INTERFACE INTERNAL I_StateInternal

PROPERTY INTERNAL _InQueue : BOOL
GET
END_GET
SET
END_SET
END_PROPERTY

PROPERTY AsIState : I_State
GET
END_GET
END_PROPERTY

METHOD CanActivate : BOOL
VAR_INPUT
END_VAR
END_METHOD

METHOD CanDeactivate : BOOL
VAR_INPUT
END_VAR
END_METHOD

METHOD OnExecute
VAR_INPUT
END_VAR
END_METHOD

METHOD OnExit
VAR_INPUT
END_VAR
END_METHOD

METHOD OnInit
VAR_INPUT
END_VAR
END_METHOD

END_INTERFACE

(* stored: Version 1.1.0.1
   Itf I_StateInternal: Id {b49468d8-74b2-4523-9a8e-300190600643}
   Folder _: Id {ea11d2f9-a8d0-4b23-897a-d4e88ba71fee}
   Folder Can: Id {6780bbc3-1843-4271-8203-ac0040ac9e3c}
   Folder On: Id {e8f03b0b-d8dc-462c-b1a1-c35c1e2a61ed}
   Property _InQueue: Id {8550ca70-63f7-455b-b1b5-7891fcc34a1c}
   Get Get: Id {5dbe6b56-3c78-4259-9af1-bcc59ffac19a}
   Set Set: Id {0fefd082-13d0-4ed6-b772-6e0ca0f9a7ef}
   Property AsIState: Id {52bd4c23-9ae7-496f-9a61-1f8649bcd48d}
   Get Get: Id {e7e14f50-c152-447d-9b6a-d41ed0aaa332}
   Method CanActivate: Id {f8f7be64-9c99-4fdf-81b1-a2add969bdf5}
   Method CanDeactivate: Id {ab838055-e4d5-46d5-a42d-ccdc9271d26a}
   Method OnExecute: Id {23860f66-3827-4c1c-aa60-c228bf755ba9}
   Method OnExit: Id {387ee35a-ce91-409e-90a2-90039f63ee69}
   Method OnInit: Id {34f20feb-a6b8-476a-ac7d-107b73173ddd} *)
